// TIA Portal V20 export
DATA_BLOCK "Data_To_Safety"   // DB20
{ S7_Optimized_Access := 'TRUE' }
// stored: MemoryReserve 100
   VAR
      Main_Valve_Arms : Bool;
      Main_Valve_Clamps : Bool;
      Tip_Hydraulic_Unit : Bool;
      Reset_ESTOPS : Bool;
      Reset_REI : Bool;
      Main_Valve_HydRolls : Bool;
   END_VAR
BEGIN
END_DATA_BLOCK
